{attribute 'qualified_only'}
{attribute 'strict'}
TYPE schudmachineToestand :
(
	startup := 0,
	automode,
	blikKlemmen,
	blikSchudden
);
END_TYPE

(* stored: Version 1.1.0.1, ProductVersion 3.1.4024.15
   DUT schudmachineToestand: Id {7e6f7e17-b319-4d79-adac-d94e04a15482} *)
